(* Logix 5000 project; controller AMP_Servo_Demo 1769-L16ER-BB1B rev 32.15; software revision 32.05; part 2 of 5 *)

ADD_ON_INSTRUCTION AMP_Home   (* revision 1.0, vendor Applied Motion Products Inc. *)
// Applied Motion - Motor Homing Methods from -4  to 35  AOI
// Help:
// This AOI Execute different Homing methods from -4 to -1 and 1 to 35. Homing method -1 to -4 use for Hard Stop Homing, For all the homing methods description check the manual on Applied Motion Products Inc. website.
VAR_IN_OUT
   Input : DINT[20]; {required}   // Drive Input Assembly
        [12]   // Digital_Outputs
        [7]   // Drive_Temperature
        [2]   // Control_Mode
        [9]   // Second_Encoder_Position
        [3]   // Status_Code
        [16]   // Analog_Input1
        [0]   // Control_Word_Received
        [17]   // Analog_Input2
        [11]   // Actual_Velocity_RPS
        [10]   // Position_Error
        [4]   // Alarm_Code
        [13]   // Digital_Inputs
        [14]   // Analog_Output1
        [15]   // Analog_Output2
        [1]   // OpCode1_Received
        [8]   // Encoder_Position
        [18]   // Torque_Limit
        [19]   // Second_Encoder_Speed
        [5]   // Supply_Voltage
        [6]   // Applied_Torque
   Output : DINT[11]; {required}   // Drive Output Assembly
        [5]   // Porifle Acceleration
        [6]   // Profile Deceleration
        [0]   // Control Word
        [7]   // Target Torque
        [4]   // Target Velocity
        [1]   // OpCode 1
        [2]   // OpCode 2
        [10]   // Reserved
        [8]   // OpCode 3
        [9]   // OpCode 4
        [3]   // Target Pos
END_VAR
VAR_INPUT
   Start : BOOL; {required}   // Home the Drive (on rising edge)
   Homing_Method : DINT; {required}   // Homing Method Number Input, -4 to 35
   Home_Speed_rps : REAL; {required}   // Homing Speed 1 rps
   Home_Speed2_rps : REAL; {required}   // Homing Speed 2 rps
   Home_Acc : REAL; {required}   // Homing Acceleration of Move (rev/s/s)
   Home_Dec : REAL; {required}   // Homing Deceleration of Move (rev/s/s)
   Homing_Offset : DINT; {required}   // Homing Offset (HO) Command Value
   Hard_Stop_Homing_Torque : INT; {required}   // Homing Current (HC) Value 0-300%
END_VAR
VAR_OUTPUT
   Sent : BOOL; {access Read Only, visible}   // Home Command has been sent to drive
   In_Progress : BOOL; {access Read Only, visible}   // Homing in progress
   Done : BOOL; {access Read Only, visible}   // Homing completed without errors - Motor is Homed
   Error : BOOL; {access Read Only, visible}   // Homing failed
   State : DINT := 10; {access Read Only}   // Internal state of progress
END_VAR
VAR
   SCL_Command : INT := 'HO';   // SCL Command Characters (always 2)
   Reg2 : DINT;   // Data / SCL Register 2
   Reg1 : DINT;   // Data / SCL Register 1
   Loc_StatusCode : AMP_Status_Word_Servo; {access None}
   Loc_Input_Assembly : AMP_Input_Assembly_Servo_v2; {access None}
   Loc_Home_ONS : BOOL;
   Loc_Command_Wait2 : TIMER := (PRE := 100); {access None}   // Timer to wait between two commands
   Loc_Command_Wait1 : TIMER := (PRE := 100); {access None}   // Timer to wait between two commands
   Loc_Command_Timeout : TIMER := (PRE := 2000); {access None}   // Timer to output fault if command is not Done
   Loc_Wait_Time : TIMER := (PRE := 200); {access None}
END_VAR

ROUTINE Logic   (* ladder *)
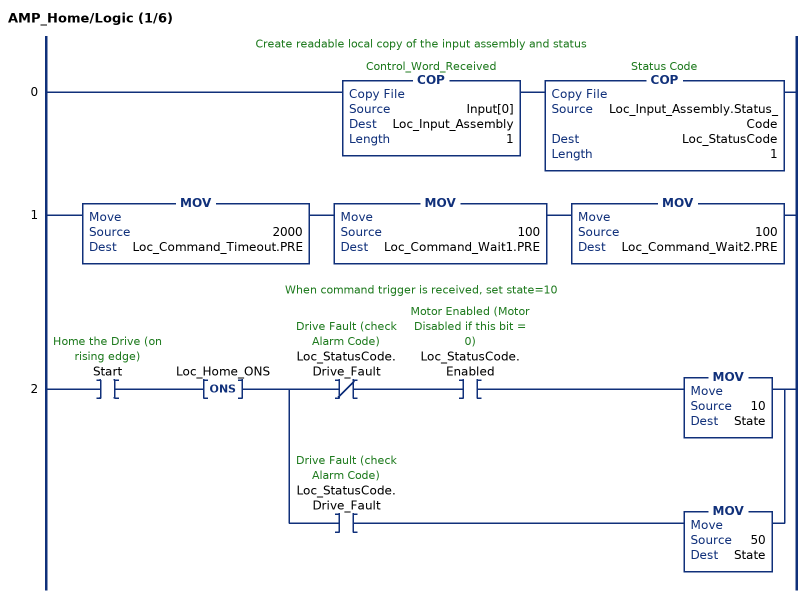
   // Create readable local copy of the input assembly and status
   0: COP(Input[0],Loc_Input_Assembly,1)COP(Loc_Input_Assembly.Status_Code,Loc_StatusCode,1);
   1: MOV(2000,Loc_Command_Timeout.PRE)MOV(100,Loc_Command_Wait1.PRE)MOV(100,Loc_Command_Wait2.PRE);
   // When command trigger is received, set state=10
   2: XIC(Start)ONS(Loc_Home_ONS)[XIO(Loc_StatusCode.Drive_Fault) XIC(Loc_StatusCode.Enabled) MOV(10,State) ,XIC(Loc_StatusCode.Drive_Fault) MOV(50,State) ];
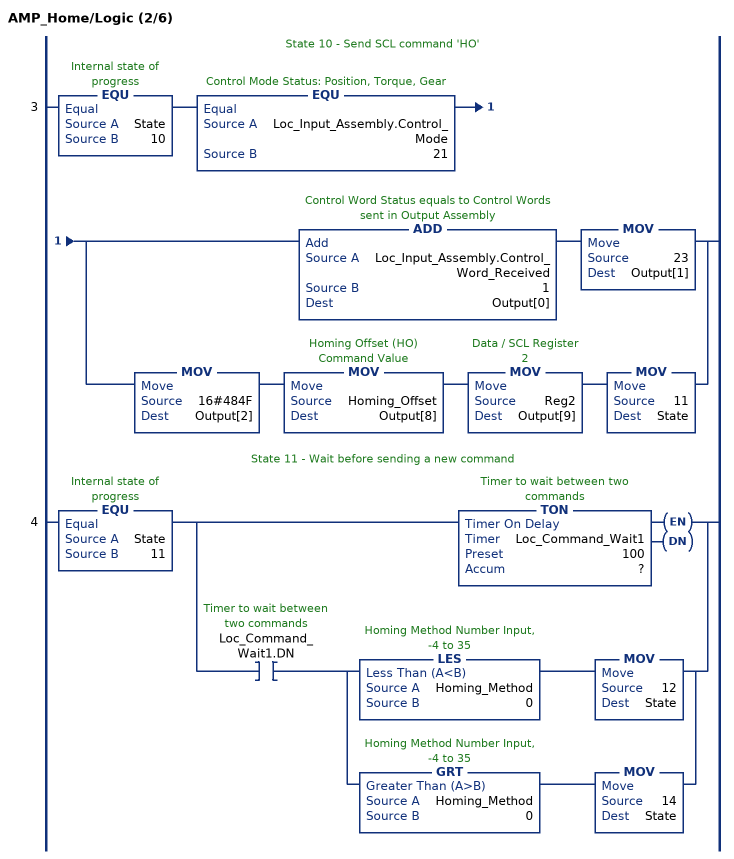
   // State 10 - Send SCL command 'HO'
   3: EQU(State,10)EQU(Loc_Input_Assembly.Control_Mode,21)[ADD(Loc_Input_Assembly.Control_Word_Received,1,Output[0]) MOV(23,Output[1]) ,MOV(16#484F,Output[2]) MOV(Homing_Offset,Output[8]) MOV(Reg2,Output[9]) MOV(11,State) ];
   // State 11 - Wait before sending a new command
   4: EQU(State,11)[TON(Loc_Command_Wait1,?,?) ,XIC(Loc_Command_Wait1.DN) [LES(Homing_Method,0) MOV(12,State) ,GRT(Homing_Method,0) MOV(14,State) ] ];
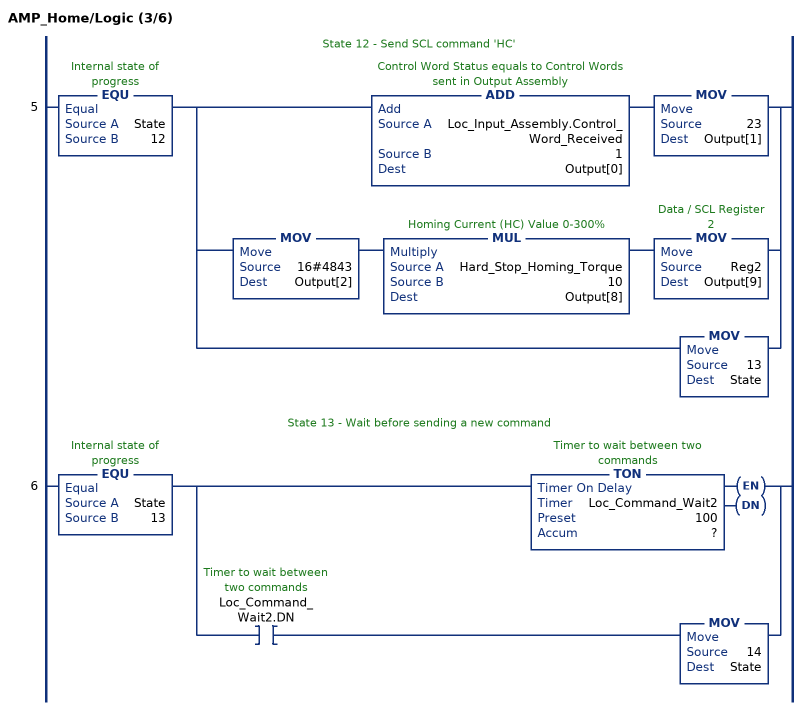
   // State 12 - Send SCL command 'HC'
   5: EQU(State,12)[ADD(Loc_Input_Assembly.Control_Word_Received,1,Output[0]) MOV(23,Output[1]) ,MOV(16#4843,Output[2]) MUL(Hard_Stop_Homing_Torque,10,Output[8]) MOV(Reg2,Output[9]) ,MOV(13,State) ];
   // State 13 - Wait before sending a new command
   6: EQU(State,13)[TON(Loc_Command_Wait2,?,?) ,XIC(Loc_Command_Wait2.DN) MOV(14,State) ];
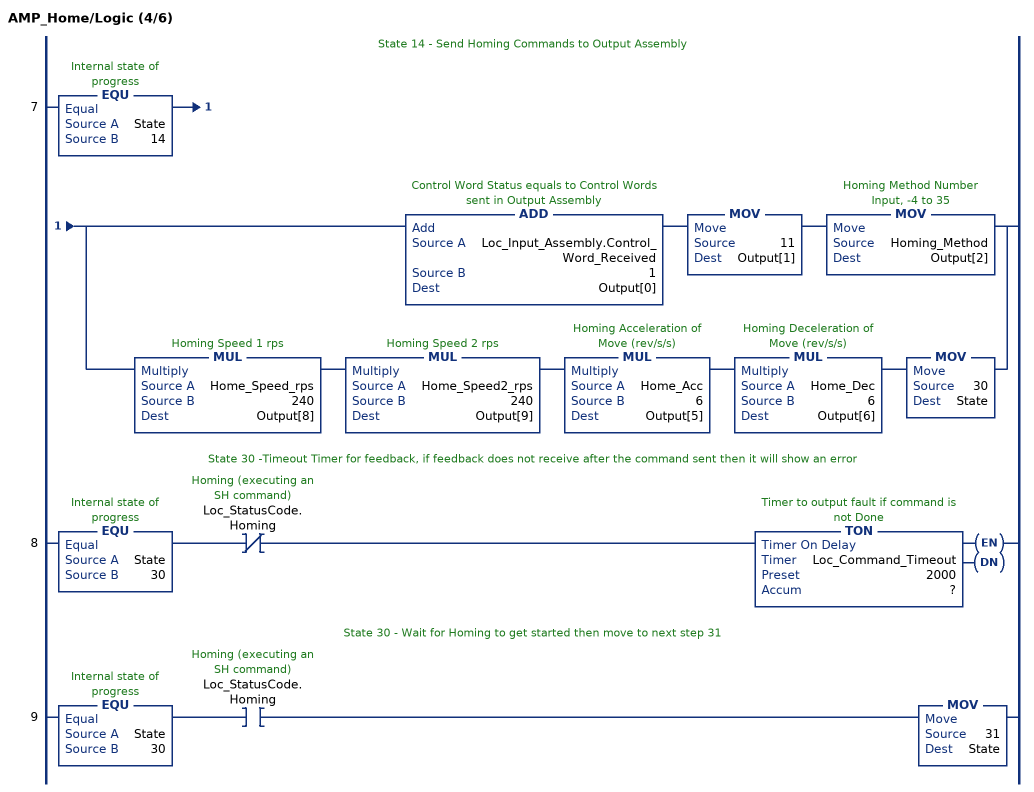
   // State 14 - Send Homing Commands to Output Assembly
   7: EQU(State,14)[ADD(Loc_Input_Assembly.Control_Word_Received,1,Output[0]) MOV(11,Output[1]) MOV(Homing_Method,Output[2]) ,MUL(Home_Speed_rps,240,Output[8]) MUL(Home_Speed2_rps,240,Output[9]) MUL(Home_Acc,6,Output[5]) MUL(Home_Dec,6,Output[6]) MOV(30,State) ];
   // State 30 -Timeout Timer for feedback, if feedback does not receive after the command sent then it will show an error
   8: EQU(State,30)XIO(Loc_StatusCode.Homing)TON(Loc_Command_Timeout,?,?);
   // State 30 - Wait for Homing to get started then move to next step 31
   9: EQU(State,30)XIC(Loc_StatusCode.Homing)MOV(31,State);
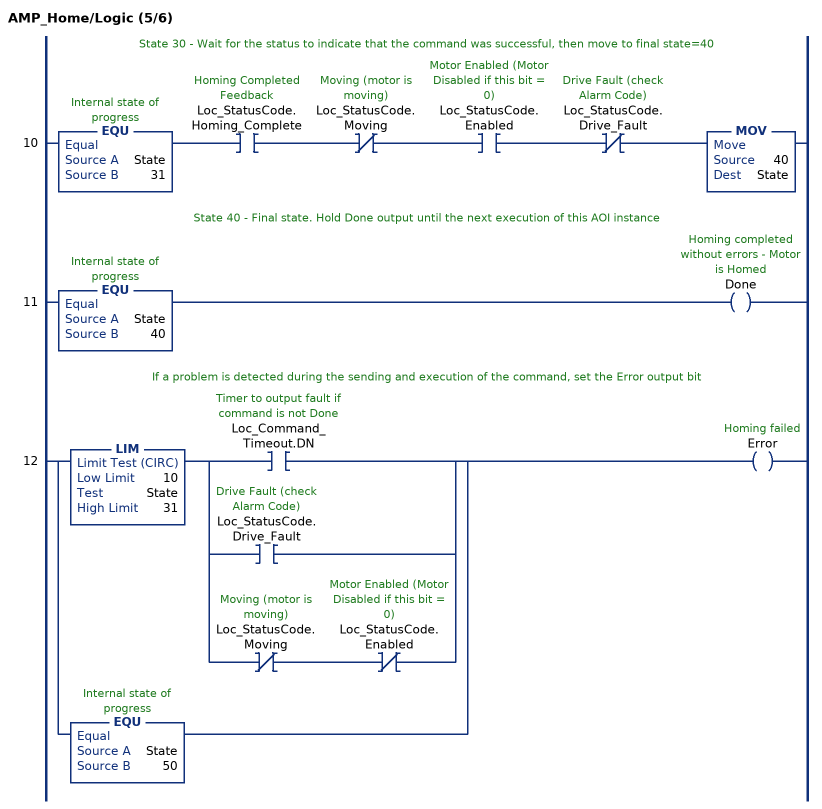
   // State 30 - Wait for the status to indicate that the command was successful, then move to final state=40
   10: EQU(State,31)XIC(Loc_StatusCode.Homing_Complete)XIO(Loc_StatusCode.Moving)XIC(Loc_StatusCode.Enabled)XIO(Loc_StatusCode.Drive_Fault)MOV(40,State);
   // State 40 - Final state. Hold Done output until the next execution of this AOI instance
   11: EQU(State,40)OTE(Done);
   // If a problem is detected during the sending and execution of the command, set the Error output bit
   12: [LIM(10,State,31) [XIC(Loc_Command_Timeout.DN) ,XIC(Loc_StatusCode.Drive_Fault) ,XIO(Loc_StatusCode.Moving) XIO(Loc_StatusCode.Enabled) ] ,EQU(State,50) ]OTE(Error);
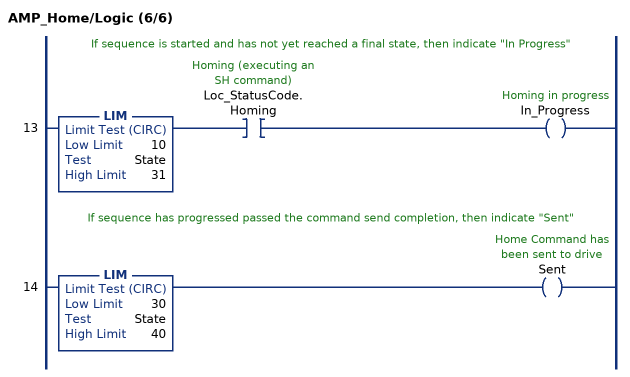
   // If sequence is started and has not yet reached a final state, then indicate "In Progress"
   13: LIM(10,State,31)XIC(Loc_StatusCode.Homing)OTE(In_Progress);
   // If sequence has progressed passed the command send completion, then indicate "Sent"
   14: LIM(30,State,40)OTE(Sent);
END_ROUTINE
END_ADD_ON_INSTRUCTION

ADD_ON_INSTRUCTION AMP_Input_Assembly   (* revision 1.0, vendor Applied Motion Products Inc. *)
// Applied Motion - Input Assembly AOI
// Help:
// The Input Assembly AOI takes raw input data from the drive and re-interprets the data, using either scaling or copying to appropriately named outputs.
VAR_IN_OUT
   Input : DINT[20]; {required}   // AMP_Assembly
   Output : AMP_Input_Assembly_Servo_v2; {required}
END_VAR
VAR_OUTPUT
   Control_Word_Received : DINT; {access Read Only, visible}   // Control Word Status equals to Control Words sent in Output Assembly
   OpCode1_Received : DINT; {access Read Only, visible}   // OpCode 1 Status equals to OpCode1 sent in Output Assembly
   Control_Mode_Active : DINT; {visible}   // Active Control Mode (0 at startup) 1= Torque, 21= Position, 10=Velocity
   Status_Code : DINT; {access Read Only, visible}   // Status Code
   Alarm_Code : DINT; {access Read Only, visible}   // Alarm Code
   DC_Bus_Voltage : REAL; {access Read Only, visible}   // DC Bus Voltage 0.1 V: ex. 242=24.2V
   Applied_Torque_Percentage : REAL; {access Read Only, visible}   // Total Applied Torque %
   Drive_Temperature_C : REAL; {access Read Only, visible}   // Drive Temperature 0.1 deg C: ex. 305=30.5 C
   Encoder_Position : DINT; {access Read Only, visible}   // Encoder Actual Position
   Position_Error : DINT; {access Read Only, visible}   // Position Error Counts
   Actual_Velocity_rps : REAL; {access Read Only, visible}   // Actual Velocity rev/sec*2: ex. 480=2 rev/sec
   Digital_Output_Status : INT; {access Read Only, visible}   // Digital Output Status
   Digital_Input_Status : INT; {access Read Only, visible}   // Digital Input Status
   Analog_Output1 : DINT; {visible}   // Analog Output 1 Value
   Analog_Output2 : DINT; {visible}   // Analog Output 2 Value
   Analog_Input_1 : DINT; {access Read Only, visible}   // Analog Input 1 Value
   Analog_Input_2 : DINT; {access Read Only, visible}   // Analog Input 2 Value
   Torque_Limit : DINT; {visible}   // Torque Limit Set Point Feedback
   External_Encoder_Position : DINT; {access Read Only, visible}   // External Encoder Position (for full closed loop servo only)
   External_Encoder_Speed_rps : DINT; {visible}   // External Encoder Speed(for full closed loop servo only)
END_VAR
VAR
   Loc_StatusCode : AMP_Status_Word_Servo; {access None}
   Loc_Input_Assembly : AMP_Input_Assembly_Servo_v2; {access None}
END_VAR

ROUTINE Logic   (* ladder *)
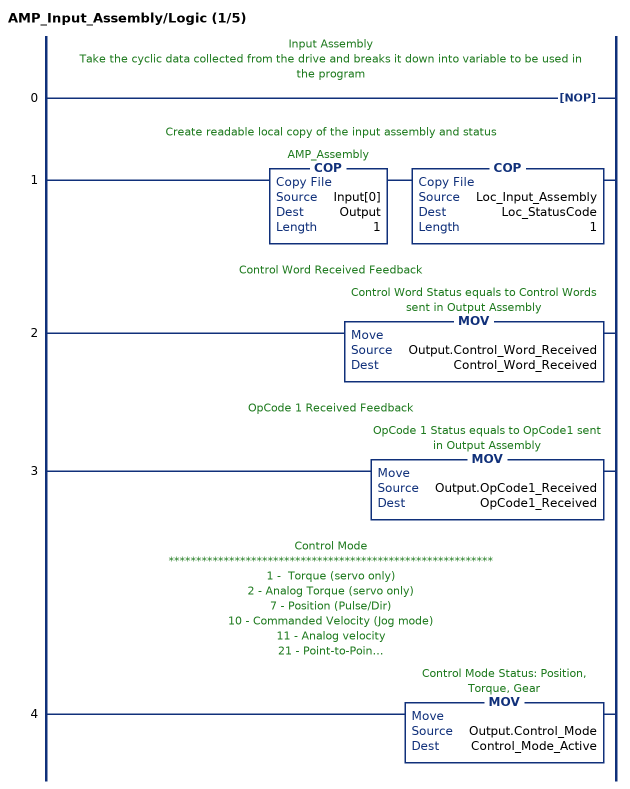
   // Input Assembly
   // Take the cyclic data collected from the drive and breaks it down into variable to be used in the program
   0: NOP();
   // Create readable local copy of the input assembly and status
   1: COP(Input[0],Output,1)COP(Loc_Input_Assembly,Loc_StatusCode,1);
   // Control Word Received Feedback
   2: MOV(Output.Control_Word_Received,Control_Word_Received);
   // OpCode 1 Received Feedback
   3: MOV(Output.OpCode1_Received,OpCode1_Received);
   // Control Mode
   // ***********************************************************
   //  1 -  Torque (servo only)
   // 2 - Analog Torque (servo only)
   // 7 - Position (Pulse/Dir)
   // 10 - Commanded Velocity (Jog mode)
   // 11 - Analog velocity
   // 21 - Point-to-Point
   // 22 - Analog Position
   4: MOV(Output.Control_Mode,Control_Mode_Active);
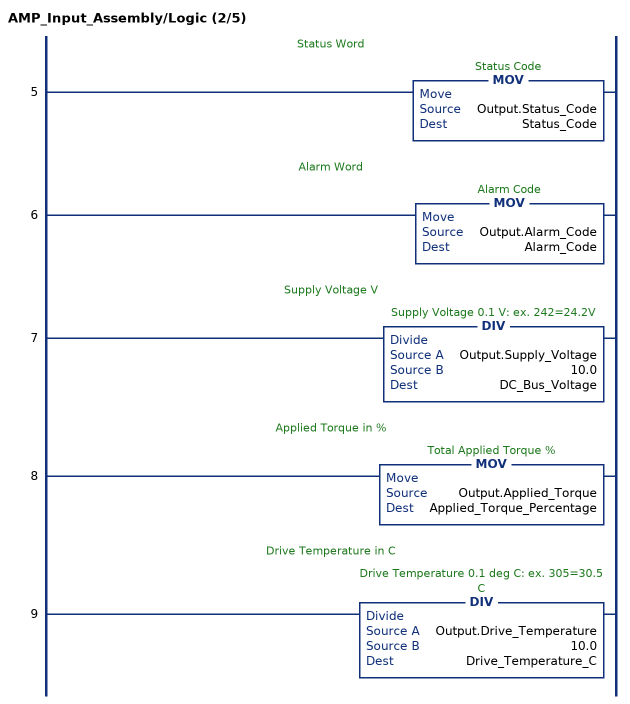
   // Status Word
   5: MOV(Output.Status_Code,Status_Code);
   // Alarm Word
   6: MOV(Output.Alarm_Code,Alarm_Code);
   // Supply Voltage V
   7: DIV(Output.Supply_Voltage,10.0,DC_Bus_Voltage);
   // Applied Torque in %
   8: MOV(Output.Applied_Torque,Applied_Torque_Percentage);
   // Drive Temperature in C
   9: DIV(Output.Drive_Temperature,10.0,Drive_Temperature_C);
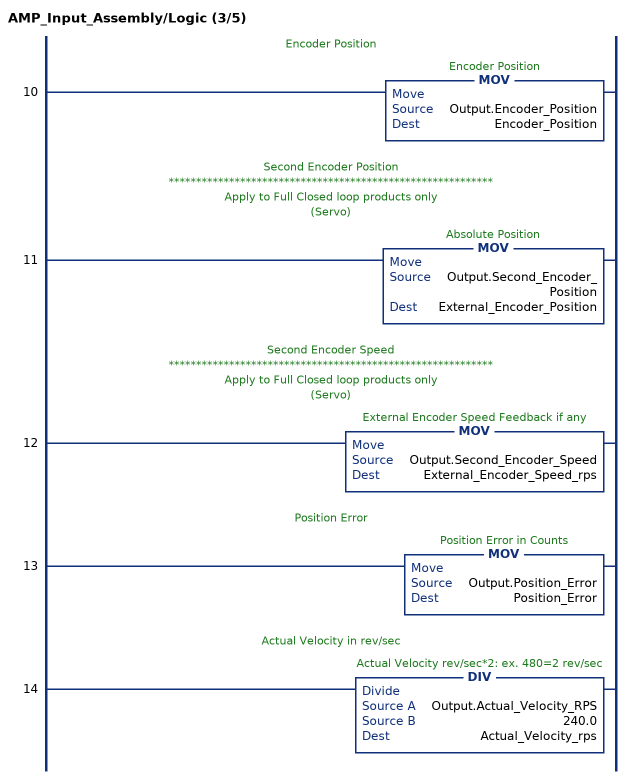
   // Encoder Position
   10: MOV(Output.Encoder_Position,Encoder_Position);
   // Second Encoder Position
   // ***********************************************************
   // Apply to Full Closed loop products only
   // (Servo)
   11: MOV(Output.Second_Encoder_Position,External_Encoder_Position);
   // Second Encoder Speed
   // ***********************************************************
   // Apply to Full Closed loop products only
   // (Servo)
   12: MOV(Output.Second_Encoder_Speed,External_Encoder_Speed_rps);
   // Position Error
   13: MOV(Output.Position_Error,Position_Error);
   // Actual Velocity in rev/sec
   14: DIV(Output.Actual_Velocity_RPS,240.0,Actual_Velocity_rps);
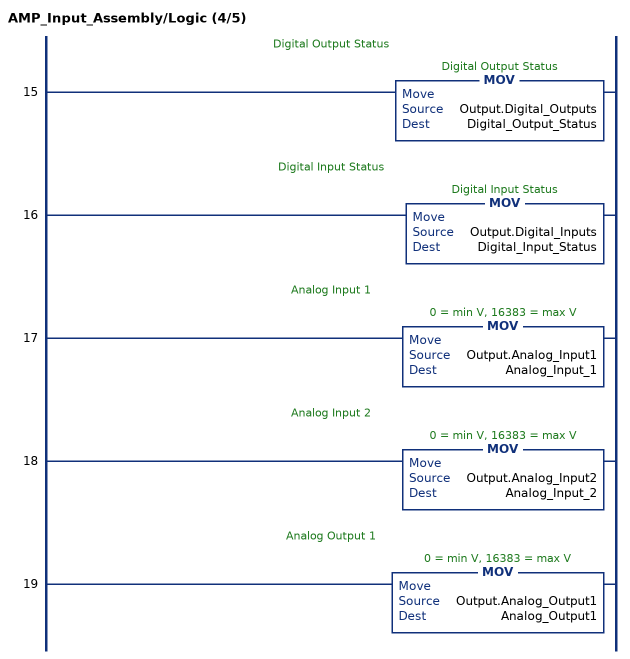
   // Digital Output Status
   15: MOV(Output.Digital_Outputs,Digital_Output_Status);
   // Digital Input Status
   16: MOV(Output.Digital_Inputs,Digital_Input_Status);
   // Analog Input 1
   17: MOV(Output.Analog_Input1,Analog_Input_1);
   // Analog Input 2
   18: MOV(Output.Analog_Input2,Analog_Input_2);
   // Analog Output 1
   19: MOV(Output.Analog_Output1,Analog_Output1);
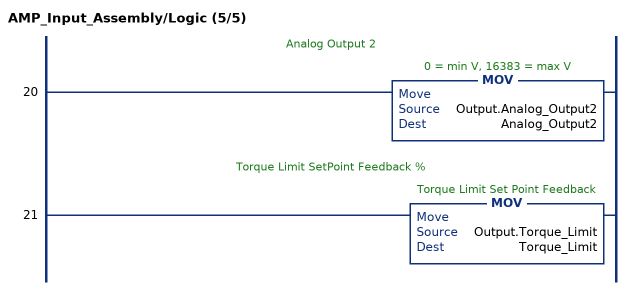
   // Analog Output 2
   20: MOV(Output.Analog_Output2,Analog_Output2);
   // Torque Limit SetPoint Feedback %
   21: MOV(Output.Torque_Limit,Torque_Limit);
END_ROUTINE
END_ADD_ON_INSTRUCTION

ADD_ON_INSTRUCTION AMP_Jog_Move   (* revision 1.0, vendor Applied Motion Products Inc. *)
// Applied Motion - Motor Jog - AOI
// Help:
// The Jog Move AOI Jog the Motor either in Positive or Negative direction(CJ). User need to use Normal Stop or Crash Stop AOI to Stop Jogging.
VAR_IN_OUT
   Input : DINT[20]; {required}   // Drive Input Assembly
        [12]   // Digital_Outputs
        [7]   // Drive_Temperature
        [2]   // Control_Mode
        [9]   // Second_Encoder_Position
        [3]   // Status_Code
        [0]   // Control_Word_Received
        [16]   // Analog_Input1
        [17]   // Analog_Input2
        [4]   // Alarm_Code
        [11]   // Actual_Velocity_RPS
        [10]   // Position_Error
        [18]   // Torque_Limit
        [13]   // Digital_Inputs
        [14]   // Analog_Output1
        [15]   // Analog_Output2
        [1]   // OpCode1_Received
        [8]   // Encoder_Position
        [5]   // Supply_Voltage
        [6]   // Applied_Torque
        [19]   // Second_Encoder_Speed
   Output : DINT[11]; {required}   // Drive Output Assembly
        [5]   // Jog Acceleration (10 rev/min/s)
        [6]   // Jog Deceleration (10 rev/min/s)
        [4]   // Jog Speed (0.25 rev/min)
        [0]   // Control Word
        [7]   // Target Torque
        [1]   // OpCode 1
        [2]   // OpCode 2
        [8]   // OpCode 3
        [9]   // OpCode 4
        [10]   // Reserved
        [3]   // Target Pos
END_VAR
VAR_INPUT
   Start : BOOL; {required}   // Jog/Move the Drive (on rising edge)
   Jog_Speed_rps : REAL; {required}   // Velocity of Jog (rev/sec)(negative=reverse)
   Jog_Acc : REAL; {required}   // Acceleration of Jog (rev/s/s)
   Jog_Dec : REAL; {required}   // Deceleration of Jog (rev/s/s)
END_VAR
VAR_OUTPUT
   Sent : BOOL; {access Read Only, visible}   // Jog Command has been sent to drive
   In_Progress : BOOL; {access Read Only, visible}   // Jog Command in progress
   Done : BOOL; {access Read Only, visible}   // Jog completed without errors - Motor Jogging
   Error : BOOL; {access Read Only, visible}   // Jog failed
   State : DINT := 10; {access Read Only}   // Internal state of progress
END_VAR
VAR
   Loc_StatusCode : AMP_Status_Word_Servo; {access None}
   Loc_Jog_ONS : BOOL;
   Loc_Input_Assembly : AMP_Input_Assembly_Servo_v2; {access None}
   Loc_Command_Timeout : TIMER := (PRE := 2000); {access None}   // Timer to output fault if command is not Done
END_VAR

ROUTINE Logic   (* ladder *)
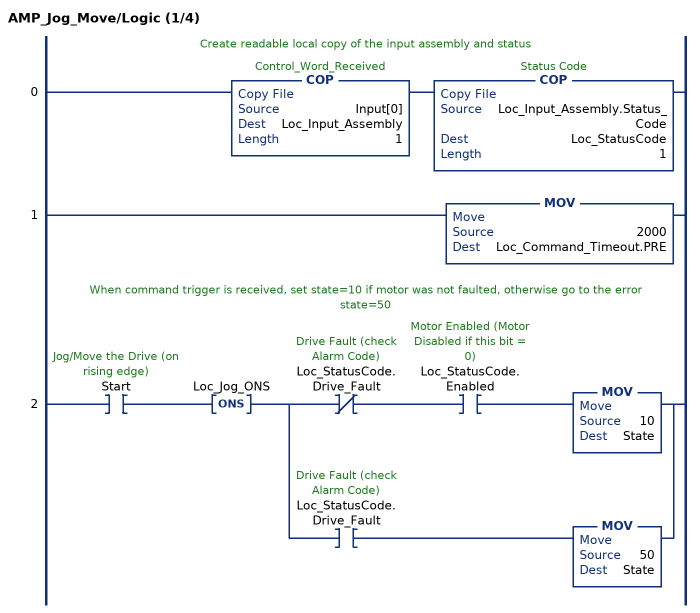
   // Create readable local copy of the input assembly and status
   0: COP(Input[0],Loc_Input_Assembly,1)COP(Loc_Input_Assembly.Status_Code,Loc_StatusCode,1);
   1: MOV(2000,Loc_Command_Timeout.PRE);
   // When command trigger is received, set state=10 if motor was not faulted, otherwise go to the error state=50
   2: XIC(Start)ONS(Loc_Jog_ONS)[XIO(Loc_StatusCode.Drive_Fault) XIC(Loc_StatusCode.Enabled) MOV(10,State) ,XIC(Loc_StatusCode.Drive_Fault) MOV(50,State) ];
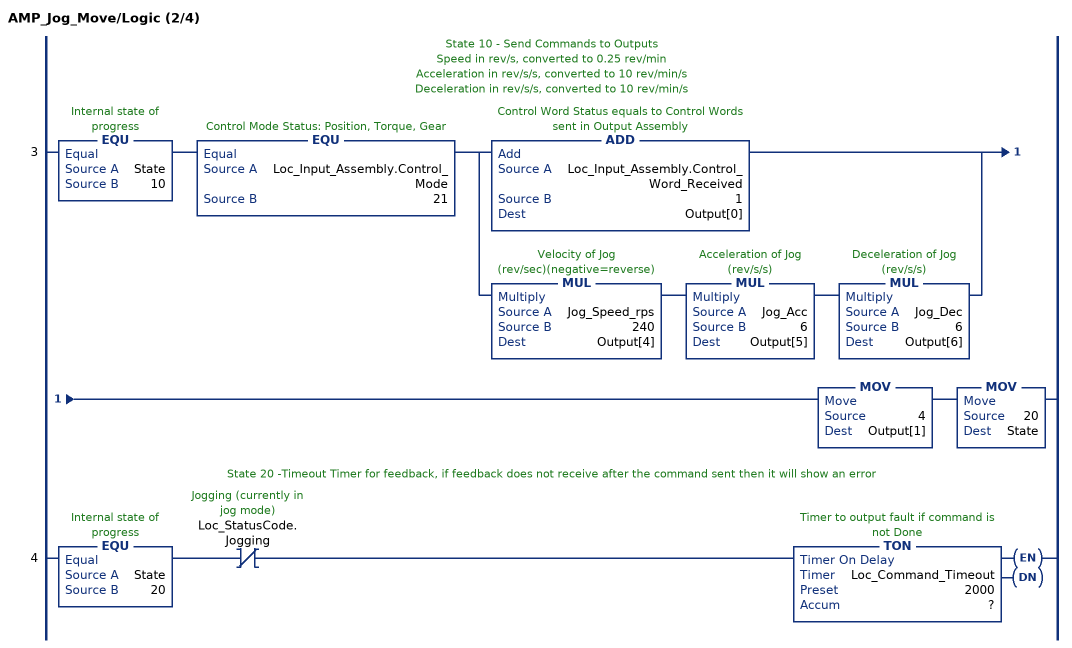
   // State 10 - Send Commands to Outputs
   // Speed in rev/s, converted to 0.25 rev/min
   // Acceleration in rev/s/s, converted to 10 rev/min/s
   // Deceleration in rev/s/s, converted to 10 rev/min/s
   3: EQU(State,10)EQU(Loc_Input_Assembly.Control_Mode,21)[ADD(Loc_Input_Assembly.Control_Word_Received,1,Output[0]) ,MUL(Jog_Speed_rps,240,Output[4]) MUL(Jog_Acc,6,Output[5]) MUL(Jog_Dec,6,Output[6]) ]MOV(4,Output[1])MOV(20,State);
   // State 20 -Timeout Timer for feedback, if feedback does not receive after the command sent then it will show an error
   4: EQU(State,20)XIO(Loc_StatusCode.Jogging)TON(Loc_Command_Timeout,?,?);
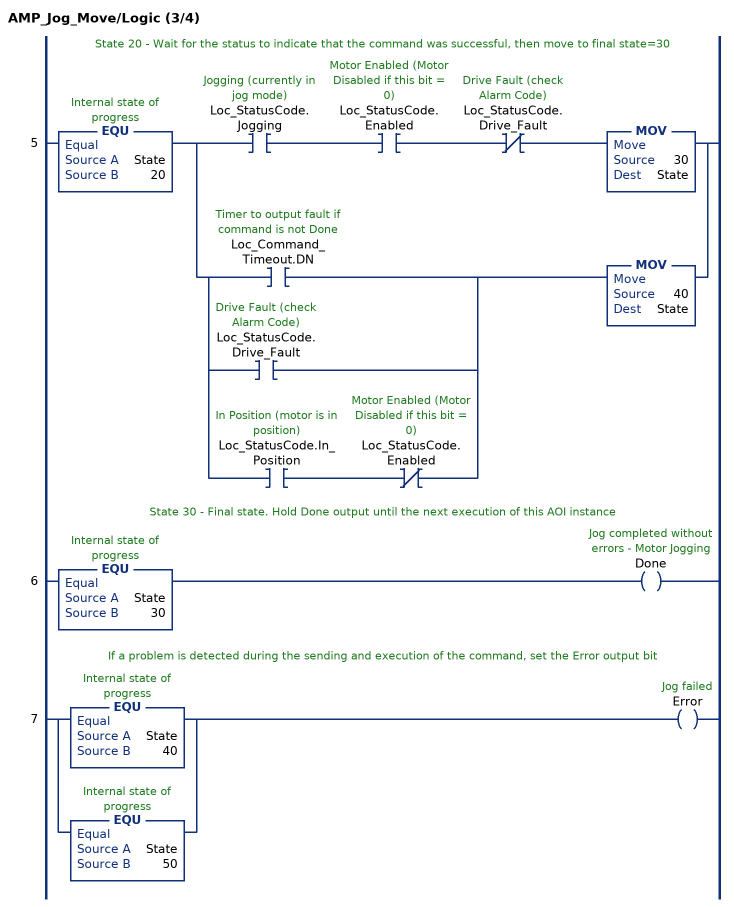
   // State 20 - Wait for the status to indicate that the command was successful, then move to final state=30
   5: EQU(State,20)[XIC(Loc_StatusCode.Jogging) XIC(Loc_StatusCode.Enabled) XIO(Loc_StatusCode.Drive_Fault) MOV(30,State) ,[XIC(Loc_Command_Timeout.DN) ,XIC(Loc_StatusCode.Drive_Fault) ,XIC(Loc_StatusCode.In_Position) XIO(Loc_StatusCode.Enabled) ] MOV(40,State) ];
   // State 30 - Final state. Hold Done output until the next execution of this AOI instance
   6: EQU(State,30)OTE(Done);
   // If a problem is detected during the sending and execution of the command, set the Error output bit
   7: [EQU(State,40) ,EQU(State,50) ]OTE(Error);
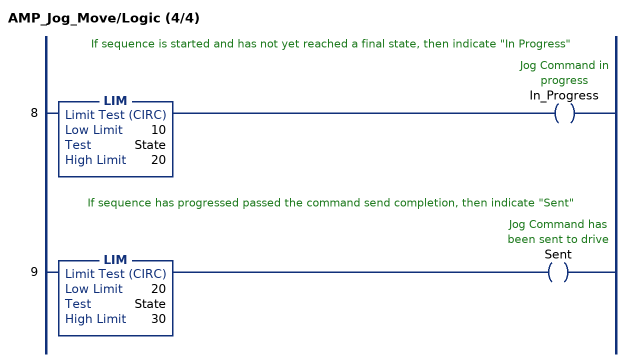
   // If sequence is started and has not yet reached a final state, then indicate "In Progress"
   8: LIM(10,State,20)OTE(In_Progress);
   // If sequence has progressed passed the command send completion, then indicate "Sent"
   9: LIM(20,State,30)OTE(Sent);
END_ROUTINE
END_ADD_ON_INSTRUCTION

ADD_ON_INSTRUCTION AMP_Motor_Disable   (* revision 1.0, vendor Applied Motion Products Inc. *)
// Applied Motion - Motor Disable - AOI
// Help:
// This AOI Disable the Motor, engage the brake if applicable(MD).
VAR_IN_OUT
   Input : DINT[20]; {required}   // Drive Input Assembly
   Output : DINT[11]; {required}   // Drive Output Assembly
        [5]   // Porifle Acceleration
        [6]   // Profile Deceleration
        [0]   // Control Word
        [7]   // Target Torque
        [1]   // OpCode 1
        [2]   // OpCode 2
        [8]   // OpCode 3
        [9]   // OpCode 4
        [4]   // Target Velocity
        [10]   // Reserved
        [3]   // Target Pos
END_VAR
VAR_INPUT
   Disable : BOOL; {required}   // Disable the Drive (on rising edge)
END_VAR
VAR_OUTPUT
   Sent : BOOL; {access Read Only, visible}   // Disable has been sent to drive
   In_Progress : BOOL; {access Read Only, visible}   // Disable in progress (not used)
   Done : BOOL; {access Read Only, visible}   // Disable completed without errors - Drive is enabled
   Error : BOOL; {access Read Only, visible}   // Disable failed
   State : DINT := 10; {access Read Only}   // Internal state of progress
END_VAR
VAR
   Loc_StatusCode : AMP_Status_Word_Servo; {access None}
   Loc_Input_Assembly : AMP_Input_Assembly_Servo_v2; {access None}
   Loc_Disable_ONS : BOOL;
   Loc_Command_Timeout : TIMER := (PRE := 2000); {access None}   // Timer to output fault if command is not Done
END_VAR

ROUTINE Logic   (* ladder *)
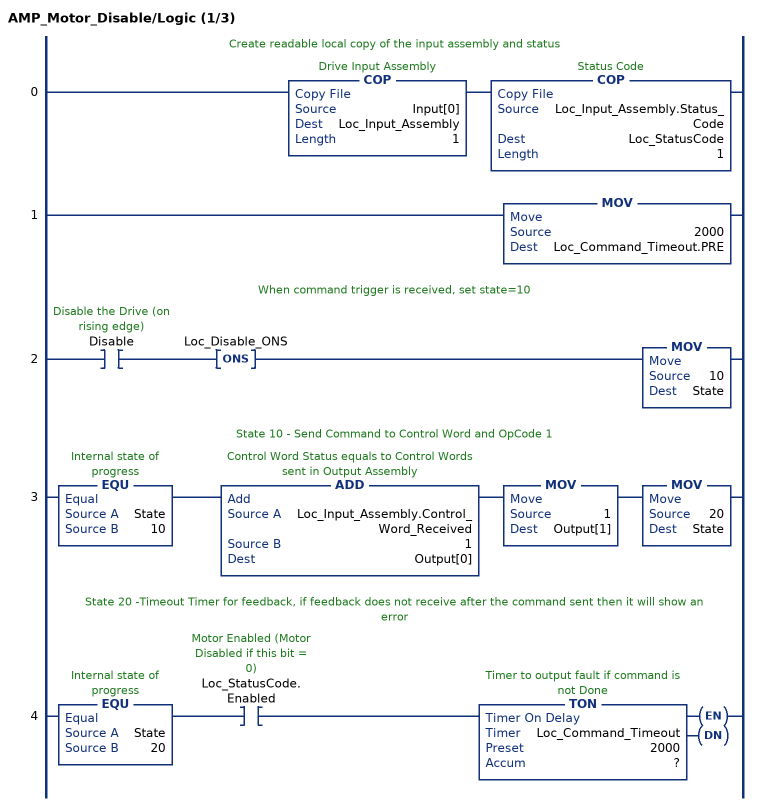
   // Create readable local copy of the input assembly and status
   0: COP(Input[0],Loc_Input_Assembly,1)COP(Loc_Input_Assembly.Status_Code,Loc_StatusCode,1);
   1: MOV(2000,Loc_Command_Timeout.PRE);
   // When command trigger is received, set state=10
   2: XIC(Disable)ONS(Loc_Disable_ONS)MOV(10,State);
   // State 10 - Send Command to Control Word and OpCode 1
   3: EQU(State,10)ADD(Loc_Input_Assembly.Control_Word_Received,1,Output[0])MOV(1,Output[1])MOV(20,State);
   // State 20 -Timeout Timer for feedback, if feedback does not receive after the command sent then it will show an error
   4: EQU(State,20)XIC(Loc_StatusCode.Enabled)TON(Loc_Command_Timeout,?,?);
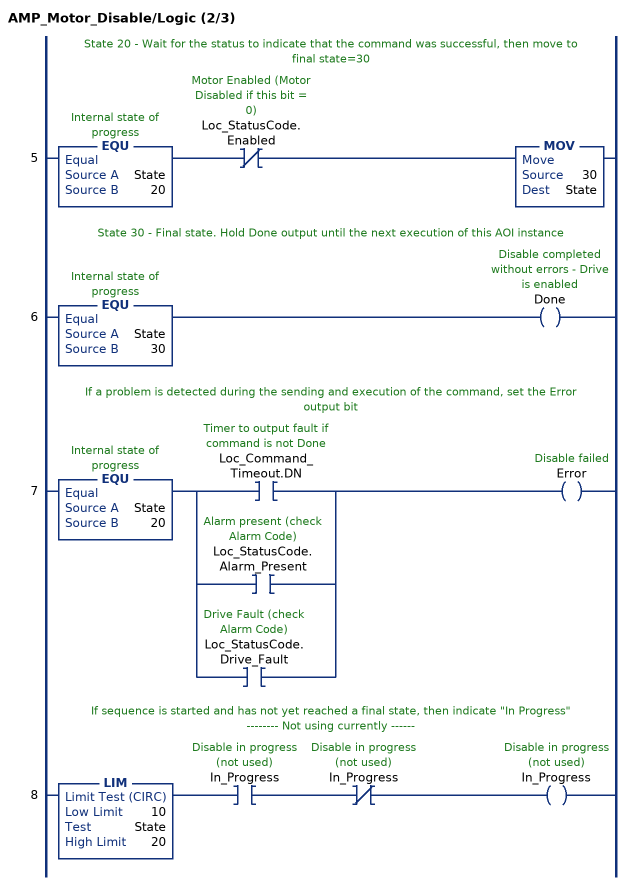
   // State 20 - Wait for the status to indicate that the command was successful, then move to final state=30
   5: EQU(State,20)XIO(Loc_StatusCode.Enabled)MOV(30,State);
   // State 30 - Final state. Hold Done output until the next execution of this AOI instance
   6: EQU(State,30)OTE(Done);
   // If a problem is detected during the sending and execution of the command, set the Error output bit
   7: EQU(State,20)[XIC(Loc_Command_Timeout.DN) ,XIC(Loc_StatusCode.Alarm_Present) ,XIC(Loc_StatusCode.Drive_Fault) ]OTE(Error);
   // If sequence is started and has not yet reached a final state, then indicate "In Progress"
   // -------- Not using currently ------
   8: LIM(10,State,20)XIC(In_Progress)XIO(In_Progress)OTE(In_Progress);
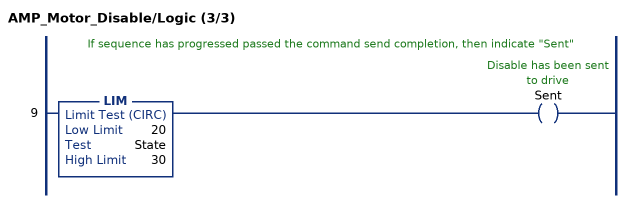
   // If sequence has progressed passed the command send completion, then indicate "Sent"
   9: LIM(20,State,30)OTE(Sent);
END_ROUTINE
END_ADD_ON_INSTRUCTION
